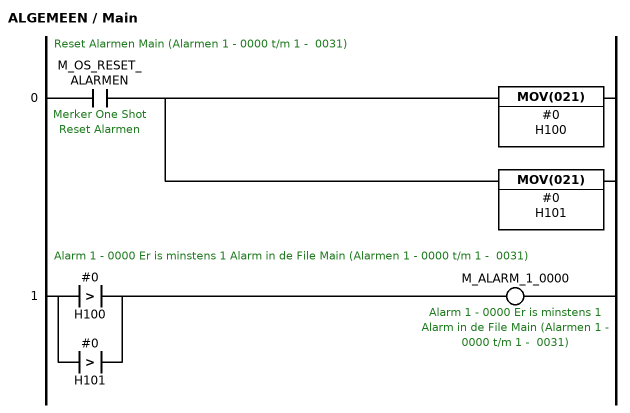
; [picture p0: ALGEMEEN / Main, rungs 0-1]
; rung 0: Reset Alarmen Main (Alarmen 1 - 0000 t/m 1 -  0031)
LD M_OS_RESET_ALARMEN  ; Merker One Shot Reset Alarmen
MOV(021) #0 H100
MOV(021) #0 H101
; rung 1: Alarm 1 - 0000 Er is minstens 1 Alarm in de File Main (Alarmen 1 - 0000 t/m 1 -  0031)
LD>(320) #0 H100
OR>(320) #0 H101
OUT M_ALARM_1_0000  ; Alarm 1 - 0000 Er is minstens 1 Alarm in de File Main (Alarmen 1 - 0000 t/m 1 -  0031)

### Section Control_Link

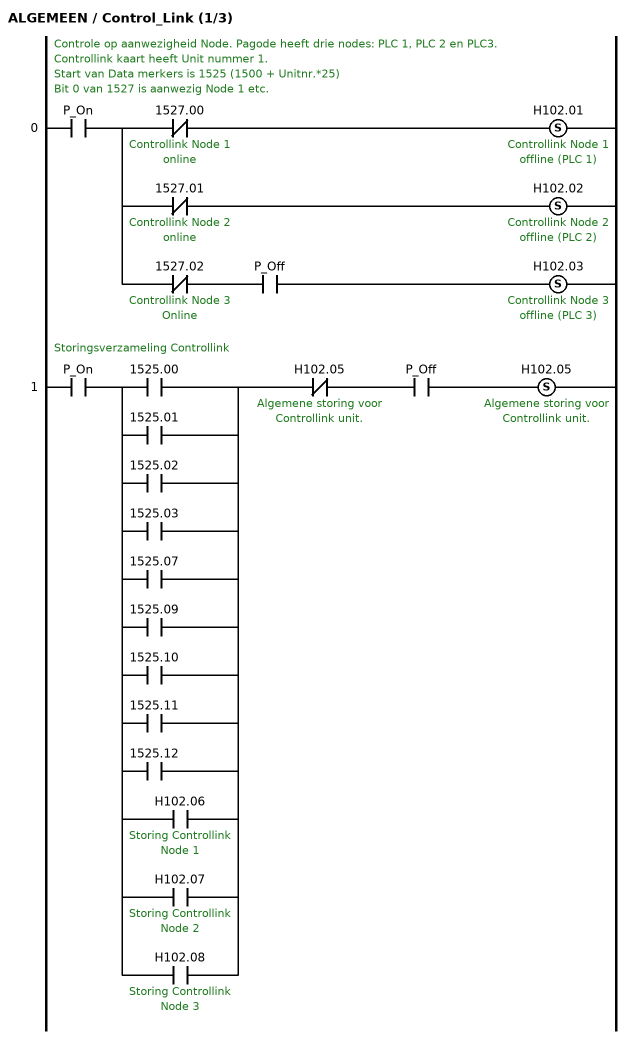
; rung 0: Controle op aanwezigheid Node. Pagode heeft drie nodes: PLC 1, PLC 2 en PLC3. / Controllink kaart heeft Unit nummer 1. / Start van Data merkers is 1525 (1500 + Unitnr.*25) / Bit 0 van 1527 is aanwezig Node 1 etc.
LD P_On
OUT TR0
ANDNOT 1527.00  ; Controllink Node 1 online
SET H102.01  ; Controllink Node 1 offline (PLC 1)
LD TR0
ANDNOT 1527.01  ; Controllink Node 2 online
SET H102.02  ; Controllink Node 2 offline (PLC 2)
LD TR0
ANDNOT 1527.02  ; Controllink Node 3 Online
AND P_Off
SET H102.03  ; Controllink Node 3 offline (PLC 3)
; rung 1: Storingsverzameling Controllink
LD P_On
LD 1525.00
OR 1525.01
OR 1525.02
OR 1525.03
OR 1525.07
OR 1525.09
OR 1525.10
OR 1525.11
OR 1525.12
OR H102.06  ; Storing Controllink Node 1
OR H102.07  ; Storing Controllink Node 2
OR H102.08  ; Storing Controllink Node 3
ANDLD
ANDNOT H102.05  ; Algemene storing voor Controllink unit.
AND P_Off
SET H102.05  ; Algemene storing voor Controllink unit.

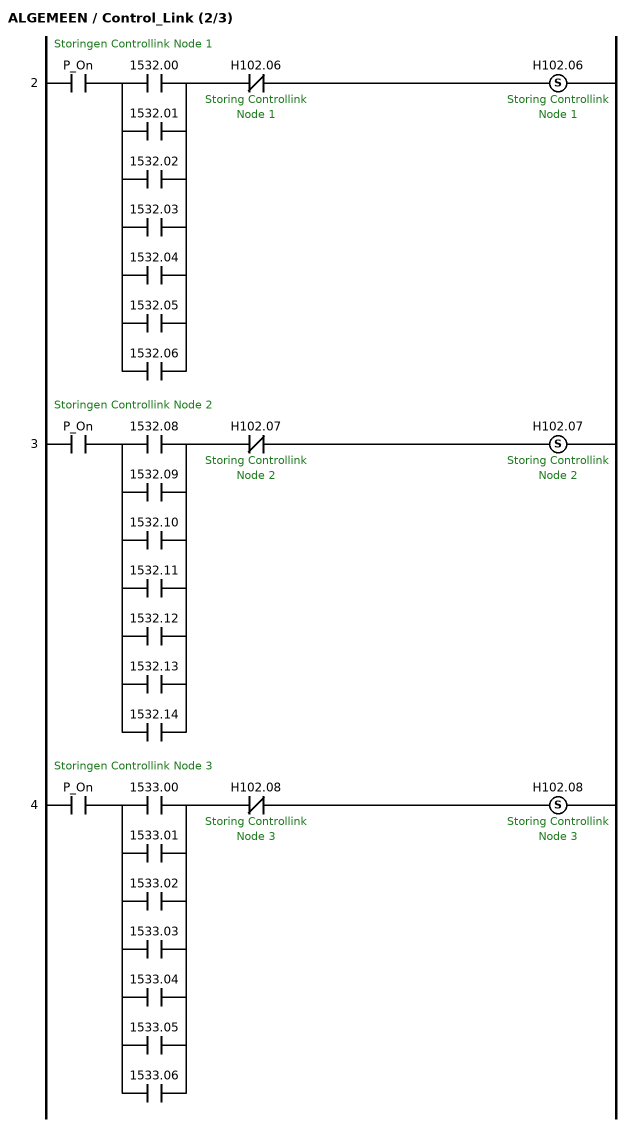
; rung 2: Storingen Controllink Node 1
LD P_On
LD 1532.00
OR 1532.01
OR 1532.02
OR 1532.03
OR 1532.04
OR 1532.05
OR 1532.06
ANDLD
ANDNOT H102.06  ; Storing Controllink Node 1
SET H102.06  ; Storing Controllink Node 1
; rung 3: Storingen Controllink Node 2
LD P_On
LD 1532.08
OR 1532.09
OR 1532.10
OR 1532.11
OR 1532.12
OR 1532.13
OR 1532.14
ANDLD
ANDNOT H102.07  ; Storing Controllink Node 2
SET H102.07  ; Storing Controllink Node 2
; rung 4: Storingen Controllink Node 3
LD P_On
LD 1533.00
OR 1533.01
OR 1533.02
OR 1533.03
OR 1533.04
OR 1533.05
OR 1533.06
ANDLD
ANDNOT H102.08  ; Storing Controllink Node 3
SET H102.08  ; Storing Controllink Node 3

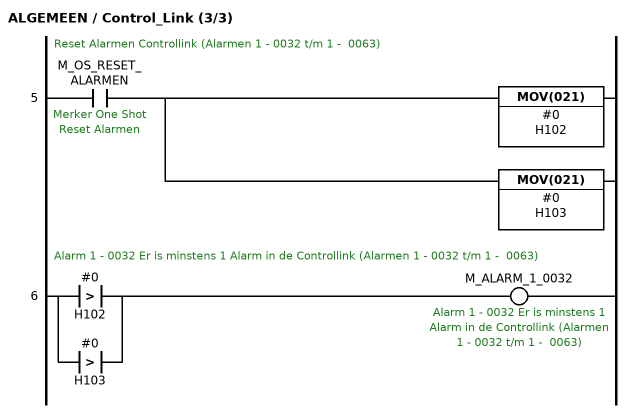
; rung 5: Reset Alarmen Controllink (Alarmen 1 - 0032 t/m 1 -  0063)
LD M_OS_RESET_ALARMEN  ; Merker One Shot Reset Alarmen
MOV(021) #0 H102
MOV(021) #0 H103
; rung 6: Alarm 1 - 0032 Er is minstens 1 Alarm in de Controllink (Alarmen 1 - 0032 t/m 1 -  0063)
LD>(320) #0 H102
OR>(320) #0 H103
OUT M_ALARM_1_0032  ; Alarm 1 - 0032 Er is minstens 1 Alarm in de Controllink (Alarmen 1 - 0032 t/m 1 -  0063)

### Section Device_Net

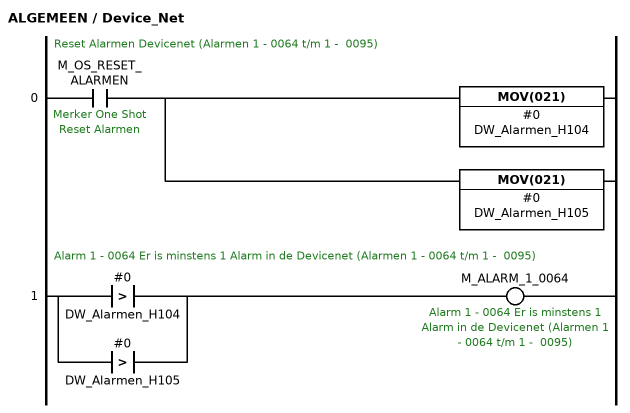
; rung 0: Reset Alarmen Devicenet (Alarmen 1 - 0064 t/m 1 -  0095)
LD M_OS_RESET_ALARMEN  ; Merker One Shot Reset Alarmen
MOV(021) #0 DW_Alarmen_H104
MOV(021) #0 DW_Alarmen_H105
; rung 1: Alarm 1 - 0064 Er is minstens 1 Alarm in de Devicenet (Alarmen 1 - 0064 t/m 1 -  0095)
LD>(320) #0 DW_Alarmen_H104
OR>(320) #0 DW_Alarmen_H105
OUT M_ALARM_1_0064  ; Alarm 1 - 0064 Er is minstens 1 Alarm in de Devicenet (Alarmen 1 - 0064 t/m 1 -  0095)

### Section Data_Opslag

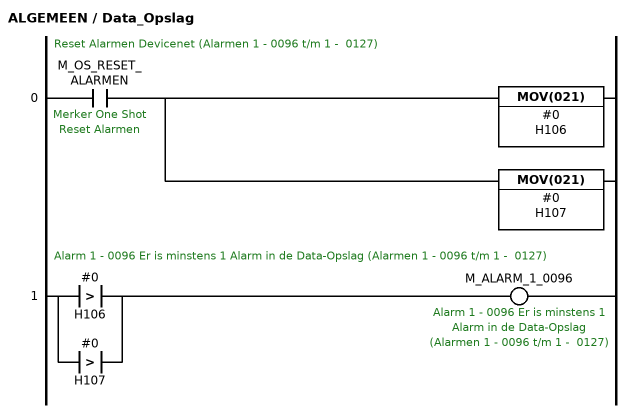
; rung 0: Reset Alarmen Devicenet (Alarmen 1 - 0096 t/m 1 -  0127)
LD M_OS_RESET_ALARMEN  ; Merker One Shot Reset Alarmen
MOV(021) #0 H106
MOV(021) #0 H107
; rung 1: Alarm 1 - 0096 Er is minstens 1 Alarm in de Data-Opslag (Alarmen 1 - 0096 t/m 1 -  0127)
LD>(320) #0 H106
OR>(320) #0 H107
OUT M_ALARM_1_0096  ; Alarm 1 - 0096 Er is minstens 1 Alarm in de Data-Opslag (Alarmen 1 - 0096 t/m 1 -  0127)

### Section Voedingen

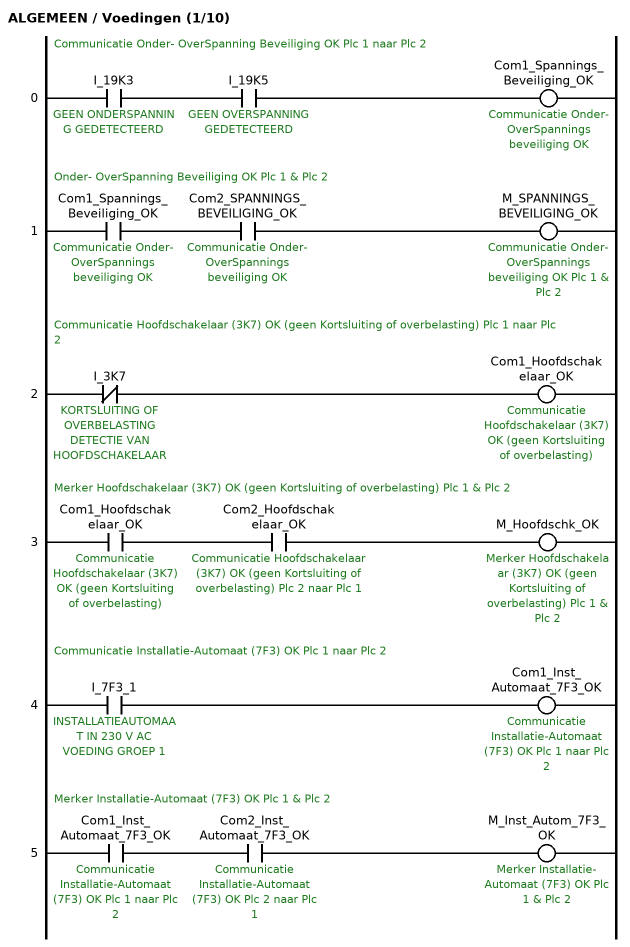
; rung 0: Communicatie Onder- OverSpanning Beveiliging OK Plc 1 naar Plc 2
LD I_19K3  ; GEEN ONDERSPANNING GEDETECTEERD
AND I_19K5  ; GEEN OVERSPANNING GEDETECTEERD
OUT Com1_Spannings_Beveiliging_OK  ; Communicatie Onder- OverSpannings beveiliging OK
; rung 1: Onder- OverSpanning Beveiliging OK Plc 1 & Plc 2
LD Com1_Spannings_Beveiliging_OK  ; Communicatie Onder- OverSpannings beveiliging OK
AND Com2_SPANNINGS_BEVEILIGING_OK  ; Communicatie Onder- OverSpannings beveiliging OK
OUT M_SPANNINGS_BEVEILIGING_OK  ; Communicatie Onder- OverSpannings beveiliging OK Plc 1 & Plc 2
; rung 2: Communicatie Hoofdschakelaar (3K7) OK (geen Kortsluiting of overbelasting) Plc 1 naar Plc 2
LDNOT I_3K7  ; KORTSLUITING OF OVERBELASTING DETECTIE VAN HOOFDSCHAKELAAR
OUT Com1_Hoofdschakelaar_OK  ; Communicatie Hoofdschakelaar (3K7) OK (geen Kortsluiting of overbelasting)
; rung 3: Merker Hoofdschakelaar (3K7) OK (geen Kortsluiting of overbelasting) Plc 1 & Plc 2
LD Com1_Hoofdschakelaar_OK  ; Communicatie Hoofdschakelaar (3K7) OK (geen Kortsluiting of overbelasting)
AND Com2_Hoofdschakelaar_OK  ; Communicatie Hoofdschakelaar (3K7) OK (geen Kortsluiting of overbelasting) Plc 2 naar Plc 1
OUT M_Hoofdschk_OK  ; Merker Hoofdschakelaar (3K7) OK (geen Kortsluiting of overbelasting) Plc 1 & Plc 2
; rung 4: Communicatie Installatie-Automaat (7F3) OK Plc 1 naar Plc 2
LD I_7F3_1  ; INSTALLATIEAUTOMAAT IN 230 V AC VOEDING GROEP 1
OUT Com1_Inst_Automaat_7F3_OK  ; Communicatie Installatie-Automaat (7F3) OK Plc 1 naar Plc 2
; rung 5: Merker Installatie-Automaat (7F3) OK Plc 1 & Plc 2
LD Com1_Inst_Automaat_7F3_OK  ; Communicatie Installatie-Automaat (7F3) OK Plc 1 naar Plc 2
AND Com2_Inst_Automaat_7F3_OK  ; Communicatie Installatie-Automaat (7F3) OK Plc 2 naar Plc 1
OUT M_Inst_Autom_7F3_OK  ; Merker Installatie-Automaat (7F3) OK Plc 1 & Plc 2

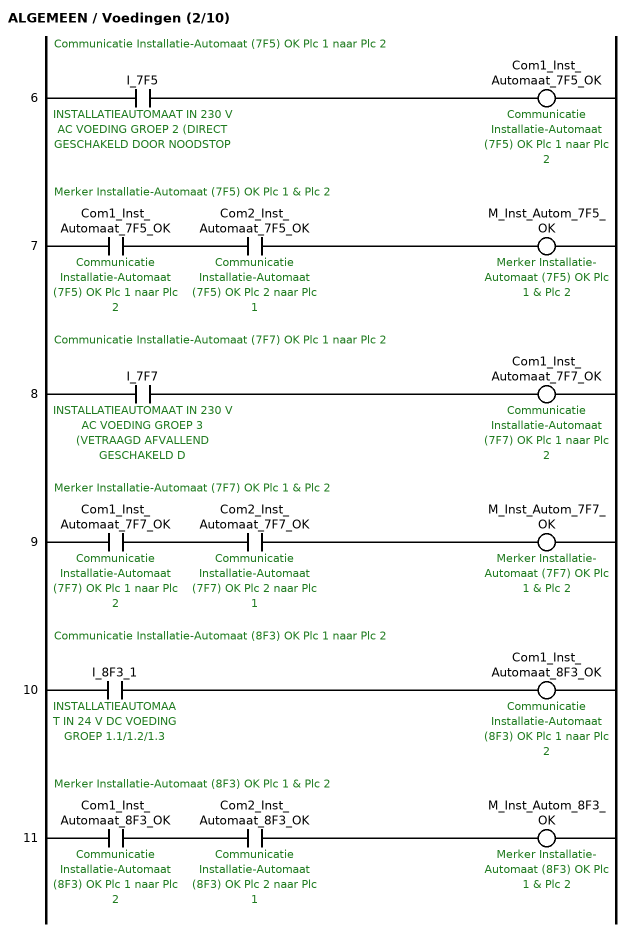
; rung 6: Communicatie Installatie-Automaat (7F5) OK Plc 1 naar Plc 2
LD I_7F5  ; INSTALLATIEAUTOMAAT IN 230 V AC VOEDING GROEP 2 (DIRECT GESCHAKELD DOOR NOODSTOP
OUT Com1_Inst_Automaat_7F5_OK  ; Communicatie Installatie-Automaat (7F5) OK Plc 1 naar Plc 2
; rung 7: Merker Installatie-Automaat (7F5) OK Plc 1 & Plc 2
LD Com1_Inst_Automaat_7F5_OK  ; Communicatie Installatie-Automaat (7F5) OK Plc 1 naar Plc 2
AND Com2_Inst_Automaat_7F5_OK  ; Communicatie Installatie-Automaat (7F5) OK Plc 2 naar Plc 1
OUT M_Inst_Autom_7F5_OK  ; Merker Installatie-Automaat (7F5) OK Plc 1 & Plc 2
; rung 8: Communicatie Installatie-Automaat (7F7) OK Plc 1 naar Plc 2
LD I_7F7  ; INSTALLATIEAUTOMAAT IN 230 V AC VOEDING GROEP 3 (VETRAAGD AFVALLEND GESCHAKELD D
OUT Com1_Inst_Automaat_7F7_OK  ; Communicatie Installatie-Automaat (7F7) OK Plc 1 naar Plc 2
; rung 9: Merker Installatie-Automaat (7F7) OK Plc 1 & Plc 2
LD Com1_Inst_Automaat_7F7_OK  ; Communicatie Installatie-Automaat (7F7) OK Plc 1 naar Plc 2
AND Com2_Inst_Automaat_7F7_OK  ; Communicatie Installatie-Automaat (7F7) OK Plc 2 naar Plc 1
OUT M_Inst_Autom_7F7_OK  ; Merker Installatie-Automaat (7F7) OK Plc 1 & Plc 2
; rung 10: Communicatie Installatie-Automaat (8F3) OK Plc 1 naar Plc 2
LD I_8F3_1  ; INSTALLATIEAUTOMAAT IN 24 V DC VOEDING GROEP 1.1/1.2/1.3
OUT Com1_Inst_Automaat_8F3_OK  ; Communicatie Installatie-Automaat (8F3) OK Plc 1 naar Plc 2
; rung 11: Merker Installatie-Automaat (8F3) OK Plc 1 & Plc 2
LD Com1_Inst_Automaat_8F3_OK  ; Communicatie Installatie-Automaat (8F3) OK Plc 1 naar Plc 2
AND Com2_Inst_Automaat_8F3_OK  ; Communicatie Installatie-Automaat (8F3) OK Plc 2 naar Plc 1
OUT M_Inst_Autom_8F3_OK  ; Merker Installatie-Automaat (8F3) OK Plc 1 & Plc 2

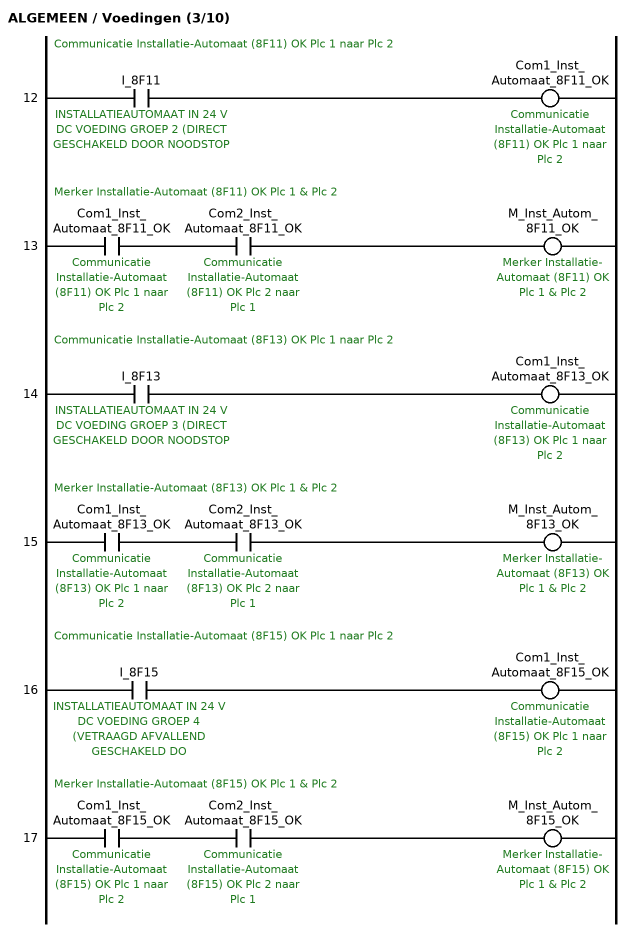
; rung 12: Communicatie Installatie-Automaat (8F11) OK Plc 1 naar Plc 2
LD I_8F11  ; INSTALLATIEAUTOMAAT IN 24 V DC VOEDING GROEP 2 (DIRECT GESCHAKELD DOOR NOODSTOP
OUT Com1_Inst_Automaat_8F11_OK  ; Communicatie Installatie-Automaat (8F11) OK Plc 1 naar Plc 2
; rung 13: Merker Installatie-Automaat (8F11) OK Plc 1 & Plc 2
LD Com1_Inst_Automaat_8F11_OK  ; Communicatie Installatie-Automaat (8F11) OK Plc 1 naar Plc 2
AND Com2_Inst_Automaat_8F11_OK  ; Communicatie Installatie-Automaat (8F11) OK Plc 2 naar Plc 1
OUT M_Inst_Autom_8F11_OK  ; Merker Installatie-Automaat (8F11) OK Plc 1 & Plc 2
; rung 14: Communicatie Installatie-Automaat (8F13) OK Plc 1 naar Plc 2
LD I_8F13  ; INSTALLATIEAUTOMAAT IN 24 V DC VOEDING GROEP 3 (DIRECT GESCHAKELD DOOR NOODSTOP
OUT Com1_Inst_Automaat_8F13_OK  ; Communicatie Installatie-Automaat (8F13) OK Plc 1 naar Plc 2
; rung 15: Merker Installatie-Automaat (8F13) OK Plc 1 & Plc 2
LD Com1_Inst_Automaat_8F13_OK  ; Communicatie Installatie-Automaat (8F13) OK Plc 1 naar Plc 2
AND Com2_Inst_Automaat_8F13_OK  ; Communicatie Installatie-Automaat (8F13) OK Plc 2 naar Plc 1
OUT M_Inst_Autom_8F13_OK  ; Merker Installatie-Automaat (8F13) OK Plc 1 & Plc 2
; rung 16: Communicatie Installatie-Automaat (8F15) OK Plc 1 naar Plc 2
LD I_8F15  ; INSTALLATIEAUTOMAAT IN 24 V DC VOEDING GROEP 4 (VETRAAGD AFVALLEND GESCHAKELD DO
OUT Com1_Inst_Automaat_8F15_OK  ; Communicatie Installatie-Automaat (8F15) OK Plc 1 naar Plc 2
; rung 17: Merker Installatie-Automaat (8F15) OK Plc 1 & Plc 2
LD Com1_Inst_Automaat_8F15_OK  ; Communicatie Installatie-Automaat (8F15) OK Plc 1 naar Plc 2
AND Com2_Inst_Automaat_8F15_OK  ; Communicatie Installatie-Automaat (8F15) OK Plc 2 naar Plc 1
OUT M_Inst_Autom_8F15_OK  ; Merker Installatie-Automaat (8F15) OK Plc 1 & Plc 2

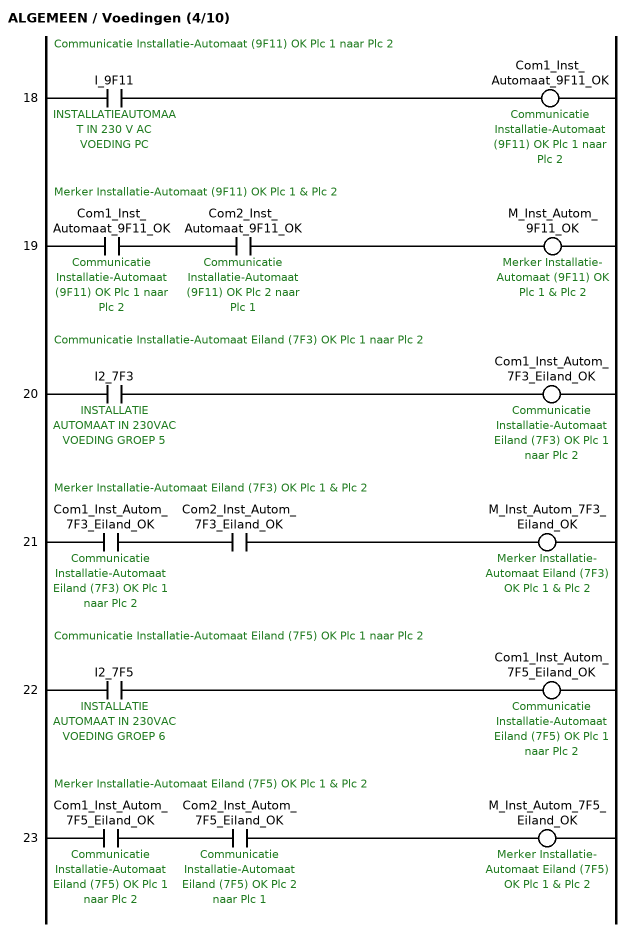
; rung 18: Communicatie Installatie-Automaat (9F11) OK Plc 1 naar Plc 2
LD I_9F11  ; INSTALLATIEAUTOMAAT IN 230 V AC VOEDING PC
OUT Com1_Inst_Automaat_9F11_OK  ; Communicatie Installatie-Automaat (9F11) OK Plc 1 naar Plc 2
; rung 19: Merker Installatie-Automaat (9F11) OK Plc 1 & Plc 2
LD Com1_Inst_Automaat_9F11_OK  ; Communicatie Installatie-Automaat (9F11) OK Plc 1 naar Plc 2
AND Com2_Inst_Automaat_9F11_OK  ; Communicatie Installatie-Automaat (9F11) OK Plc 2 naar Plc 1
OUT M_Inst_Autom_9F11_OK  ; Merker Installatie-Automaat (9F11) OK Plc 1 & Plc 2
; rung 20: Communicatie Installatie-Automaat Eiland (7F3) OK Plc 1 naar Plc 2
LD I2_7F3  ; INSTALLATIE AUTOMAAT IN 230VAC VOEDING GROEP 5
OUT Com1_Inst_Autom_7F3_Eiland_OK  ; Communicatie Installatie-Automaat Eiland (7F3) OK Plc 1 naar Plc 2
; rung 21: Merker Installatie-Automaat Eiland (7F3) OK Plc 1 & Plc 2
LD Com1_Inst_Autom_7F3_Eiland_OK  ; Communicatie Installatie-Automaat Eiland (7F3) OK Plc 1 naar Plc 2
AND Com2_Inst_Autom_7F3_Eiland_OK
OUT M_Inst_Autom_7F3_Eiland_OK  ; Merker Installatie-Automaat Eiland (7F3) OK Plc 1 & Plc 2
; rung 22: Communicatie Installatie-Automaat Eiland (7F5) OK Plc 1 naar Plc 2
LD I2_7F5  ; INSTALLATIE AUTOMAAT IN 230VAC VOEDING GROEP 6
OUT Com1_Inst_Autom_7F5_Eiland_OK  ; Communicatie Installatie-Automaat Eiland (7F5) OK Plc 1 naar Plc 2
; rung 23: Merker Installatie-Automaat Eiland (7F5) OK Plc 1 & Plc 2
LD Com1_Inst_Autom_7F5_Eiland_OK  ; Communicatie Installatie-Automaat Eiland (7F5) OK Plc 1 naar Plc 2
AND Com2_Inst_Autom_7F5_Eiland_OK  ; Communicatie Installatie-Automaat Eiland (7F5) OK Plc 2 naar Plc 1
OUT M_Inst_Autom_7F5_Eiland_OK  ; Merker Installatie-Automaat Eiland (7F5) OK Plc 1 & Plc 2

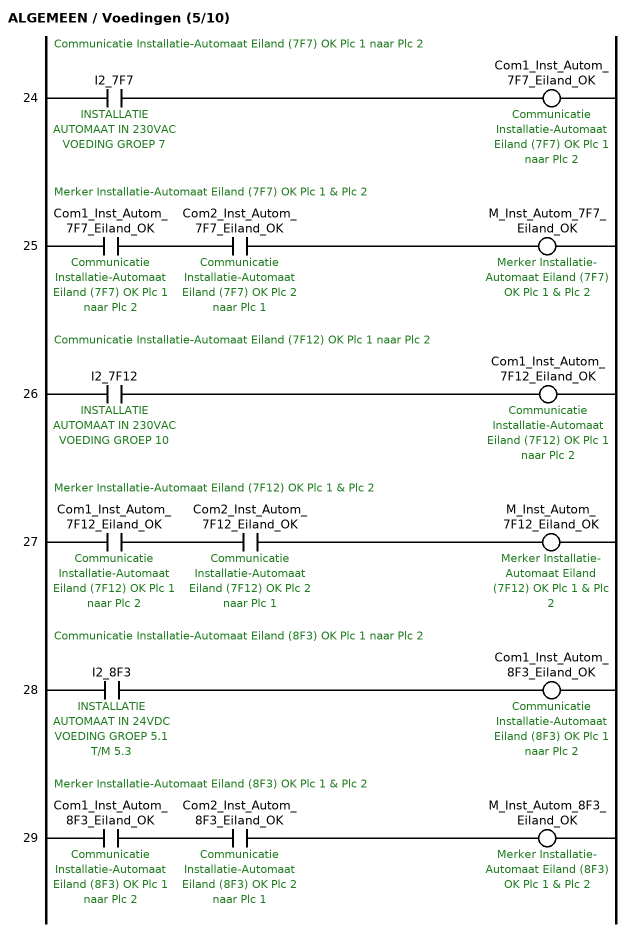
; rung 24: Communicatie Installatie-Automaat Eiland (7F7) OK Plc 1 naar Plc 2
LD I2_7F7  ; INSTALLATIE AUTOMAAT IN 230VAC VOEDING GROEP 7
OUT Com1_Inst_Autom_7F7_Eiland_OK  ; Communicatie Installatie-Automaat Eiland (7F7) OK Plc 1 naar Plc 2
; rung 25: Merker Installatie-Automaat Eiland (7F7) OK Plc 1 & Plc 2
LD Com1_Inst_Autom_7F7_Eiland_OK  ; Communicatie Installatie-Automaat Eiland (7F7) OK Plc 1 naar Plc 2
AND Com2_Inst_Autom_7F7_Eiland_OK  ; Communicatie Installatie-Automaat Eiland (7F7) OK Plc 2 naar Plc 1
OUT M_Inst_Autom_7F7_Eiland_OK  ; Merker Installatie-Automaat Eiland (7F7) OK Plc 1 & Plc 2
; rung 26: Communicatie Installatie-Automaat Eiland (7F12) OK Plc 1 naar Plc 2
LD I2_7F12  ; INSTALLATIE AUTOMAAT IN 230VAC VOEDING GROEP 10
OUT Com1_Inst_Autom_7F12_Eiland_OK  ; Communicatie Installatie-Automaat Eiland (7F12) OK Plc 1 naar Plc 2
; rung 27: Merker Installatie-Automaat Eiland (7F12) OK Plc 1 & Plc 2
LD Com1_Inst_Autom_7F12_Eiland_OK  ; Communicatie Installatie-Automaat Eiland (7F12) OK Plc 1 naar Plc 2
AND Com2_Inst_Autom_7F12_Eiland_OK  ; Communicatie Installatie-Automaat Eiland (7F12) OK Plc 2 naar Plc 1
OUT M_Inst_Autom_7F12_Eiland_OK  ; Merker Installatie-Automaat Eiland (7F12) OK Plc 1 & Plc 2
; rung 28: Communicatie Installatie-Automaat Eiland (8F3) OK Plc 1 naar Plc 2
LD I2_8F3  ; INSTALLATIE AUTOMAAT IN 24VDC VOEDING GROEP 5.1 T/M 5.3
OUT Com1_Inst_Autom_8F3_Eiland_OK  ; Communicatie Installatie-Automaat Eiland (8F3) OK Plc 1 naar Plc 2
; rung 29: Merker Installatie-Automaat Eiland (8F3) OK Plc 1 & Plc 2
LD Com1_Inst_Autom_8F3_Eiland_OK  ; Communicatie Installatie-Automaat Eiland (8F3) OK Plc 1 naar Plc 2
AND Com2_Inst_Autom_8F3_Eiland_OK  ; Communicatie Installatie-Automaat Eiland (8F3) OK Plc 2 naar Plc 1
OUT M_Inst_Autom_8F3_Eiland_OK  ; Merker Installatie-Automaat Eiland (8F3) OK Plc 1 & Plc 2

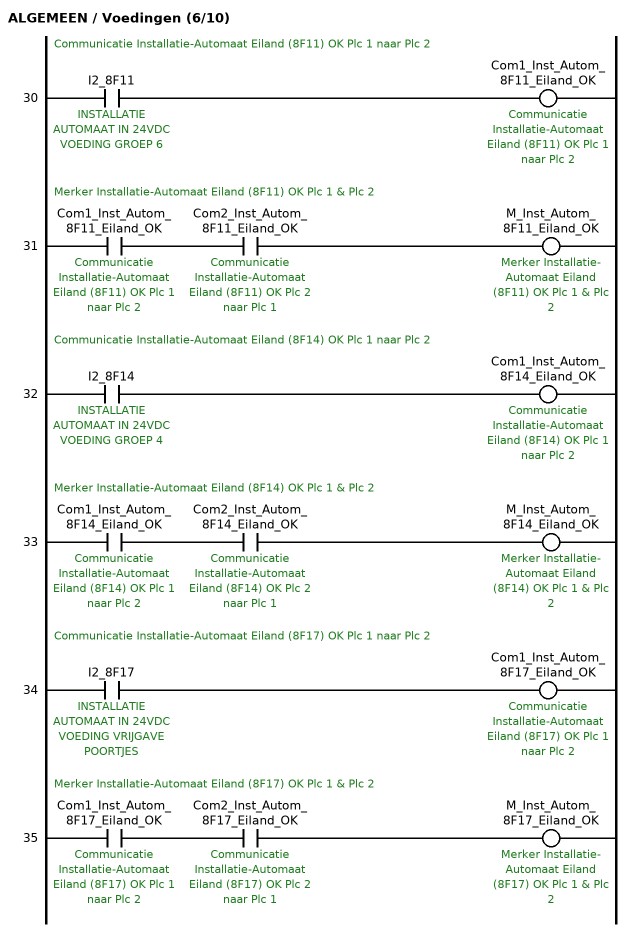
; rung 30: Communicatie Installatie-Automaat Eiland (8F11) OK Plc 1 naar Plc 2
LD I2_8F11  ; INSTALLATIE AUTOMAAT IN 24VDC VOEDING GROEP 6
OUT Com1_Inst_Autom_8F11_Eiland_OK  ; Communicatie Installatie-Automaat Eiland (8F11) OK Plc 1 naar Plc 2
; rung 31: Merker Installatie-Automaat Eiland (8F11) OK Plc 1 & Plc 2
LD Com1_Inst_Autom_8F11_Eiland_OK  ; Communicatie Installatie-Automaat Eiland (8F11) OK Plc 1 naar Plc 2
AND Com2_Inst_Autom_8F11_Eiland_OK  ; Communicatie Installatie-Automaat Eiland (8F11) OK Plc 2 naar Plc 1
OUT M_Inst_Autom_8F11_Eiland_OK  ; Merker Installatie-Automaat Eiland (8F11) OK Plc 1 & Plc 2
; rung 32: Communicatie Installatie-Automaat Eiland (8F14) OK Plc 1 naar Plc 2
LD I2_8F14  ; INSTALLATIE AUTOMAAT IN 24VDC VOEDING GROEP 4
OUT Com1_Inst_Autom_8F14_Eiland_OK  ; Communicatie Installatie-Automaat Eiland (8F14) OK Plc 1 naar Plc 2
; rung 33: Merker Installatie-Automaat Eiland (8F14) OK Plc 1 & Plc 2
LD Com1_Inst_Autom_8F14_Eiland_OK  ; Communicatie Installatie-Automaat Eiland (8F14) OK Plc 1 naar Plc 2
AND Com2_Inst_Autom_8F14_Eiland_OK  ; Communicatie Installatie-Automaat Eiland (8F14) OK Plc 2 naar Plc 1
OUT M_Inst_Autom_8F14_Eiland_OK  ; Merker Installatie-Automaat Eiland (8F14) OK Plc 1 & Plc 2
; rung 34: Communicatie Installatie-Automaat Eiland (8F17) OK Plc 1 naar Plc 2
LD I2_8F17  ; INSTALLATIE AUTOMAAT IN 24VDC VOEDING VRIJGAVE POORTJES
OUT Com1_Inst_Autom_8F17_Eiland_OK  ; Communicatie Installatie-Automaat Eiland (8F17) OK Plc 1 naar Plc 2
; rung 35: Merker Installatie-Automaat Eiland (8F17) OK Plc 1 & Plc 2
LD Com1_Inst_Autom_8F17_Eiland_OK  ; Communicatie Installatie-Automaat Eiland (8F17) OK Plc 1 naar Plc 2
AND Com2_Inst_Autom_8F17_Eiland_OK  ; Communicatie Installatie-Automaat Eiland (8F17) OK Plc 2 naar Plc 1
OUT M_Inst_Autom_8F17_Eiland_OK  ; Merker Installatie-Automaat Eiland (8F17) OK Plc 1 & Plc 2

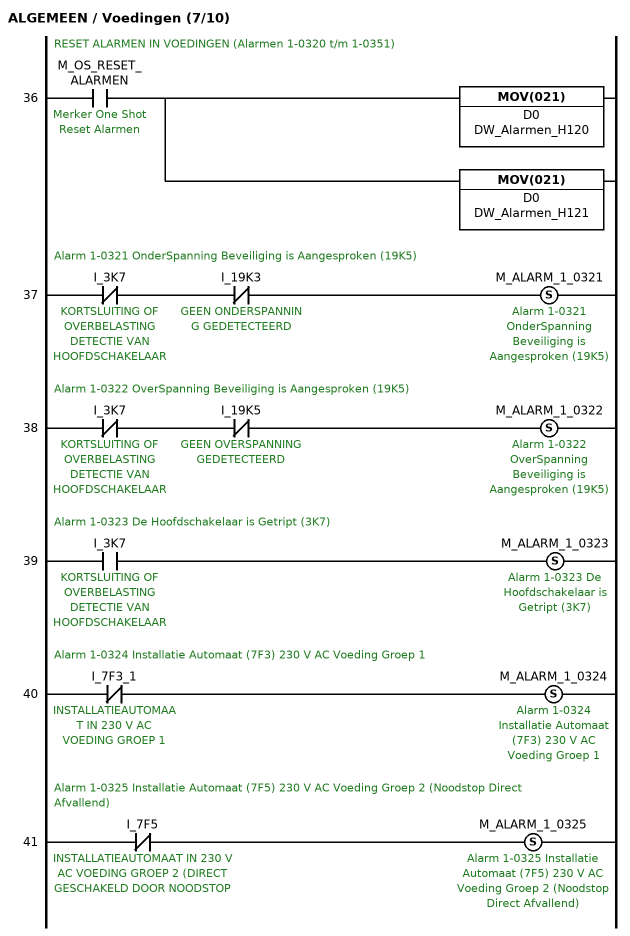
; rung 36: RESET ALARMEN IN VOEDINGEN (Alarmen 1-0320 t/m 1-0351)
LD M_OS_RESET_ALARMEN  ; Merker One Shot Reset Alarmen
MOV(021) D0 DW_Alarmen_H120
MOV(021) D0 DW_Alarmen_H121
; rung 37: Alarm 1-0321 OnderSpanning Beveiliging is Aangesproken (19K5)
LDNOT I_3K7  ; KORTSLUITING OF OVERBELASTING DETECTIE VAN HOOFDSCHAKELAAR
ANDNOT I_19K3  ; GEEN ONDERSPANNING GEDETECTEERD
SET M_ALARM_1_0321  ; Alarm 1-0321 OnderSpanning Beveiliging is Aangesproken (19K5)
; rung 38: Alarm 1-0322 OverSpanning Beveiliging is Aangesproken (19K5)
LDNOT I_3K7  ; KORTSLUITING OF OVERBELASTING DETECTIE VAN HOOFDSCHAKELAAR
ANDNOT I_19K5  ; GEEN OVERSPANNING GEDETECTEERD
SET M_ALARM_1_0322  ; Alarm 1-0322 OverSpanning Beveiliging is Aangesproken (19K5)
; rung 39: Alarm 1-0323 De Hoofdschakelaar is Getript (3K7)
LD I_3K7  ; KORTSLUITING OF OVERBELASTING DETECTIE VAN HOOFDSCHAKELAAR
SET M_ALARM_1_0323  ; Alarm 1-0323 De Hoofdschakelaar is Getript (3K7)
; rung 40: Alarm 1-0324 Installatie Automaat (7F3) 230 V AC Voeding Groep 1
LDNOT I_7F3_1  ; INSTALLATIEAUTOMAAT IN 230 V AC VOEDING GROEP 1
SET M_ALARM_1_0324  ; Alarm 1-0324 Installatie Automaat (7F3) 230 V AC Voeding Groep 1
; rung 41: Alarm 1-0325 Installatie Automaat (7F5) 230 V AC Voeding Groep 2 (Noodstop Direct Afvallend)
LDNOT I_7F5  ; INSTALLATIEAUTOMAAT IN 230 V AC VOEDING GROEP 2 (DIRECT GESCHAKELD DOOR NOODSTOP
SET M_ALARM_1_0325  ; Alarm 1-0325 Installatie Automaat (7F5) 230 V AC Voeding Groep 2 (Noodstop Direct Afvallend)

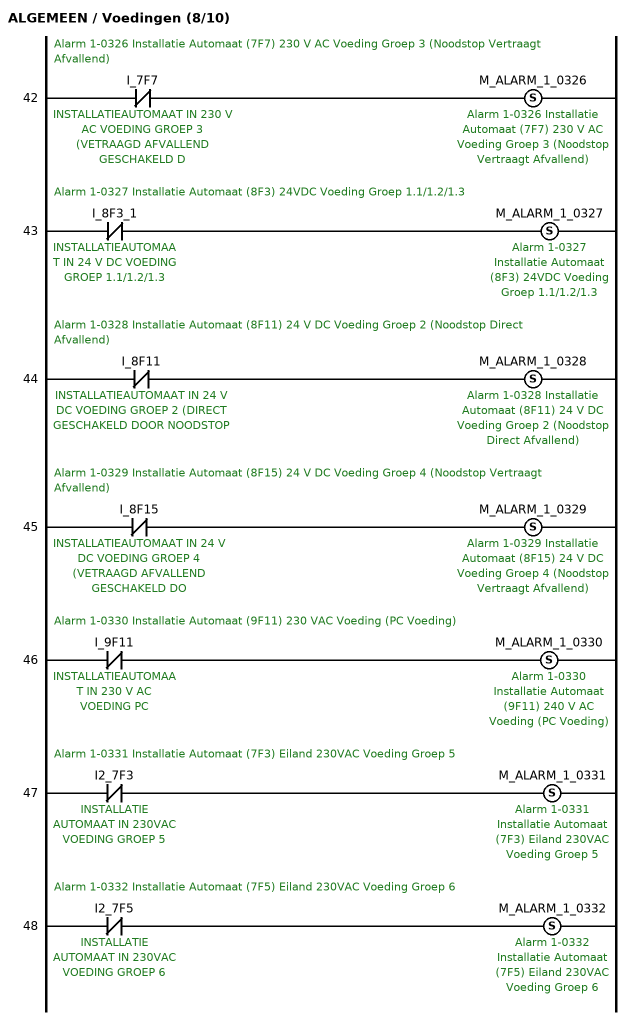
; rung 42: Alarm 1-0326 Installatie Automaat (7F7) 230 V AC Voeding Groep 3 (Noodstop Vertraagt Afvallend)
LDNOT I_7F7  ; INSTALLATIEAUTOMAAT IN 230 V AC VOEDING GROEP 3 (VETRAAGD AFVALLEND GESCHAKELD D
SET M_ALARM_1_0326  ; Alarm 1-0326 Installatie Automaat (7F7) 230 V AC Voeding Groep 3 (Noodstop Vertraagt Afvallend)
; rung 43: Alarm 1-0327 Installatie Automaat (8F3) 24VDC Voeding Groep 1.1/1.2/1.3
LDNOT I_8F3_1  ; INSTALLATIEAUTOMAAT IN 24 V DC VOEDING GROEP 1.1/1.2/1.3
SET M_ALARM_1_0327  ; Alarm 1-0327 Installatie Automaat (8F3) 24VDC Voeding Groep 1.1/1.2/1.3
; rung 44: Alarm 1-0328 Installatie Automaat (8F11) 24 V DC Voeding Groep 2 (Noodstop Direct Afvallend)
LDNOT I_8F11  ; INSTALLATIEAUTOMAAT IN 24 V DC VOEDING GROEP 2 (DIRECT GESCHAKELD DOOR NOODSTOP
SET M_ALARM_1_0328  ; Alarm 1-0328 Installatie Automaat (8F11) 24 V DC Voeding Groep 2 (Noodstop Direct Afvallend)
; rung 45: Alarm 1-0329 Installatie Automaat (8F15) 24 V DC Voeding Groep 4 (Noodstop Vertraagt Afvallend)
LDNOT I_8F15  ; INSTALLATIEAUTOMAAT IN 24 V DC VOEDING GROEP 4 (VETRAAGD AFVALLEND GESCHAKELD DO
SET M_ALARM_1_0329  ; Alarm 1-0329 Installatie Automaat (8F15) 24 V DC Voeding Groep 4 (Noodstop Vertraagt Afvallend)
; rung 46: Alarm 1-0330 Installatie Automaat (9F11) 230 VAC Voeding (PC Voeding)
LDNOT I_9F11  ; INSTALLATIEAUTOMAAT IN 230 V AC VOEDING PC
SET M_ALARM_1_0330  ; Alarm 1-0330 Installatie Automaat (9F11) 240 V AC Voeding (PC Voeding)
; rung 47: Alarm 1-0331 Installatie Automaat (7F3) Eiland 230VAC Voeding Groep 5
LDNOT I2_7F3  ; INSTALLATIE AUTOMAAT IN 230VAC VOEDING GROEP 5
SET M_ALARM_1_0331  ; Alarm 1-0331 Installatie Automaat (7F3) Eiland 230VAC Voeding Groep 5
; rung 48: Alarm 1-0332 Installatie Automaat (7F5) Eiland 230VAC Voeding Groep 6
LDNOT I2_7F5  ; INSTALLATIE AUTOMAAT IN 230VAC VOEDING GROEP 6
SET M_ALARM_1_0332  ; Alarm 1-0332 Installatie Automaat (7F5) Eiland 230VAC Voeding Groep 6

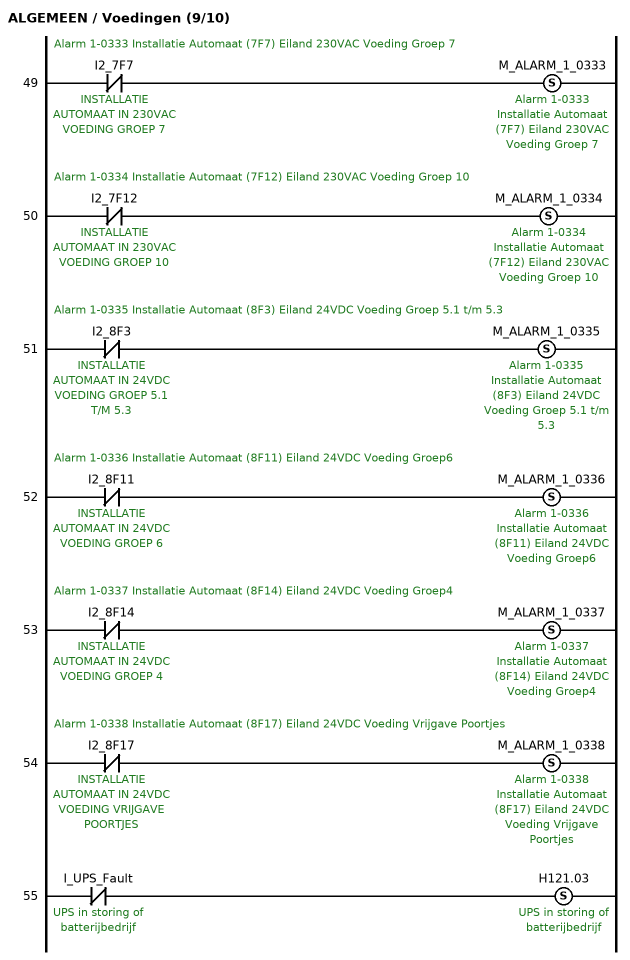
; rung 49: Alarm 1-0333 Installatie Automaat (7F7) Eiland 230VAC Voeding Groep 7
LDNOT I2_7F7  ; INSTALLATIE AUTOMAAT IN 230VAC VOEDING GROEP 7
SET M_ALARM_1_0333  ; Alarm 1-0333 Installatie Automaat (7F7) Eiland 230VAC Voeding Groep 7
; rung 50: Alarm 1-0334 Installatie Automaat (7F12) Eiland 230VAC Voeding Groep 10
LDNOT I2_7F12  ; INSTALLATIE AUTOMAAT IN 230VAC VOEDING GROEP 10
SET M_ALARM_1_0334  ; Alarm 1-0334 Installatie Automaat (7F12) Eiland 230VAC Voeding Groep 10
; rung 51: Alarm 1-0335 Installatie Automaat (8F3) Eiland 24VDC Voeding Groep 5.1 t/m 5.3
LDNOT I2_8F3  ; INSTALLATIE AUTOMAAT IN 24VDC VOEDING GROEP 5.1 T/M 5.3
SET M_ALARM_1_0335  ; Alarm 1-0335 Installatie Automaat (8F3) Eiland 24VDC Voeding Groep 5.1 t/m 5.3
; rung 52: Alarm 1-0336 Installatie Automaat (8F11) Eiland 24VDC Voeding Groep6
LDNOT I2_8F11  ; INSTALLATIE AUTOMAAT IN 24VDC VOEDING GROEP 6
SET M_ALARM_1_0336  ; Alarm 1-0336 Installatie Automaat (8F11) Eiland 24VDC Voeding Groep6
; rung 53: Alarm 1-0337 Installatie Automaat (8F14) Eiland 24VDC Voeding Groep4
LDNOT I2_8F14  ; INSTALLATIE AUTOMAAT IN 24VDC VOEDING GROEP 4
SET M_ALARM_1_0337  ; Alarm 1-0337 Installatie Automaat (8F14) Eiland 24VDC Voeding Groep4
; rung 54: Alarm 1-0338 Installatie Automaat (8F17) Eiland 24VDC Voeding Vrijgave Poortjes
LDNOT I2_8F17  ; INSTALLATIE AUTOMAAT IN 24VDC VOEDING VRIJGAVE POORTJES
SET M_ALARM_1_0338  ; Alarm 1-0338 Installatie Automaat (8F17) Eiland 24VDC Voeding Vrijgave Poortjes
; rung 55
LDNOT I_UPS_Fault  ; UPS in storing of batterijbedrijf
SET H121.03  ; UPS in storing of batterijbedrijf

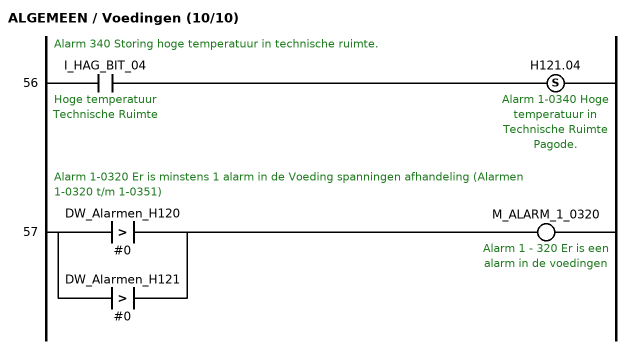
; rung 56: Alarm 340 Storing hoge temperatuur in technische ruimte.
LD I_HAG_BIT_04  ; Hoge temperatuur Technische Ruimte
SET H121.04  ; Alarm 1-0340 Hoge temperatuur in Technische Ruimte Pagode.
; rung 57: Alarm 1-0320 Er is minstens 1 alarm in de Voeding spanningen afhandeling (Alarmen 1-0320 t/m 1-0351)
LD>(320) DW_Alarmen_H120 #0
OR>(320) DW_Alarmen_H121 #0
OUT M_ALARM_1_0320  ; Alarm 1 - 320 Er is een alarm in de voedingen

### Section I_O_Controle

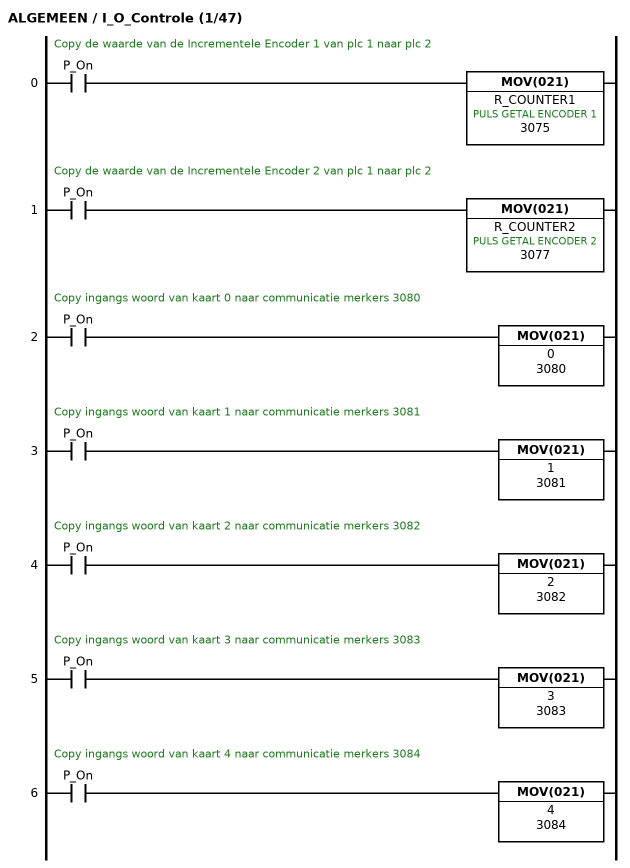
; rung 0: Copy de waarde van de Incrementele Encoder 1 van plc 1 naar plc 2
LD P_On
MOV(021) R_COUNTER1 3075  ; PULS GETAL ENCODER 1
; rung 1: Copy de waarde van de Incrementele Encoder 2 van plc 1 naar plc 2
LD P_On
MOV(021) R_COUNTER2 3077  ; PULS GETAL ENCODER 2
; rung 2: Copy ingangs woord van kaart 0 naar communicatie merkers 3080
LD P_On
MOV(021) 0 3080
; rung 3: Copy ingangs woord van kaart 1 naar communicatie merkers 3081
LD P_On
MOV(021) 1 3081
; rung 4: Copy ingangs woord van kaart 2 naar communicatie merkers 3082
LD P_On
MOV(021) 2 3082
; rung 5: Copy ingangs woord van kaart 3 naar communicatie merkers 3083
LD P_On
MOV(021) 3 3083
; rung 6: Copy ingangs woord van kaart 4 naar communicatie merkers 3084
LD P_On
MOV(021) 4 3084

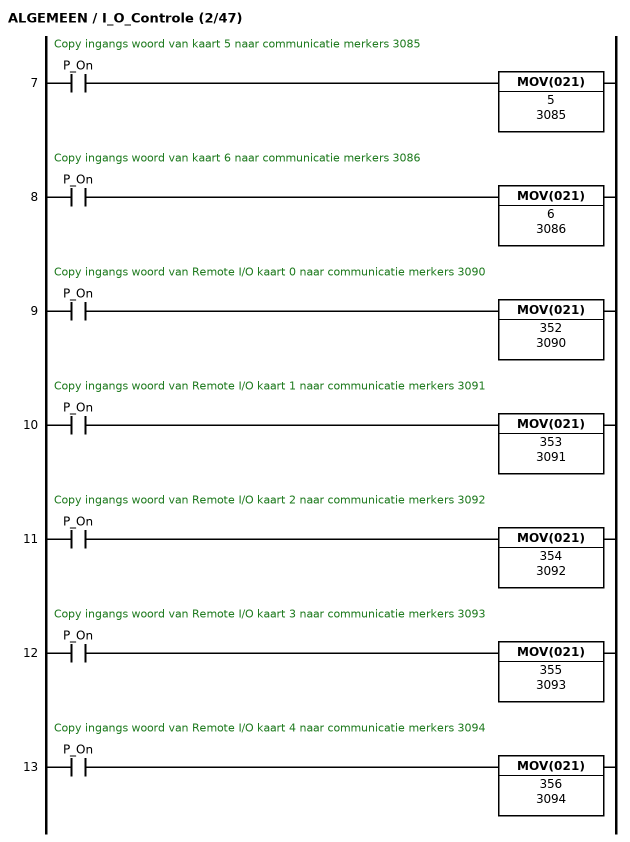
; rung 7: Copy ingangs woord van kaart 5 naar communicatie merkers 3085
LD P_On
MOV(021) 5 3085
; rung 8: Copy ingangs woord van kaart 6 naar communicatie merkers 3086
LD P_On
MOV(021) 6 3086
; rung 9: Copy ingangs woord van Remote I/O kaart 0 naar communicatie merkers 3090
LD P_On
MOV(021) 352 3090
; rung 10: Copy ingangs woord van Remote I/O kaart 1 naar communicatie merkers 3091
LD P_On
MOV(021) 353 3091
; rung 11: Copy ingangs woord van Remote I/O kaart 2 naar communicatie merkers 3092
LD P_On
MOV(021) 354 3092
; rung 12: Copy ingangs woord van Remote I/O kaart 3 naar communicatie merkers 3093
LD P_On
MOV(021) 355 3093
; rung 13: Copy ingangs woord van Remote I/O kaart 4 naar communicatie merkers 3094
LD P_On
MOV(021) 356 3094

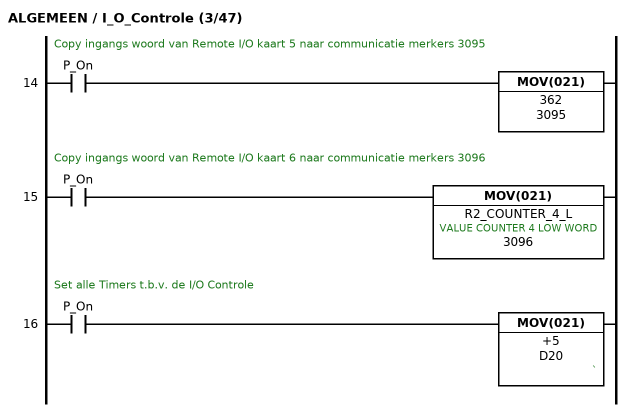
; rung 14: Copy ingangs woord van Remote I/O kaart 5 naar communicatie merkers 3095
LD P_On
MOV(021) 362 3095
; rung 15: Copy ingangs woord van Remote I/O kaart 6 naar communicatie merkers 3096
LD P_On
MOV(021) R2_COUNTER_4_L 3096  ; VALUE COUNTER 4 LOW WORD
; rung 16: Set alle Timers t.b.v. de I/O Controle
LD P_On
MOV(021) +5 D20  ; `

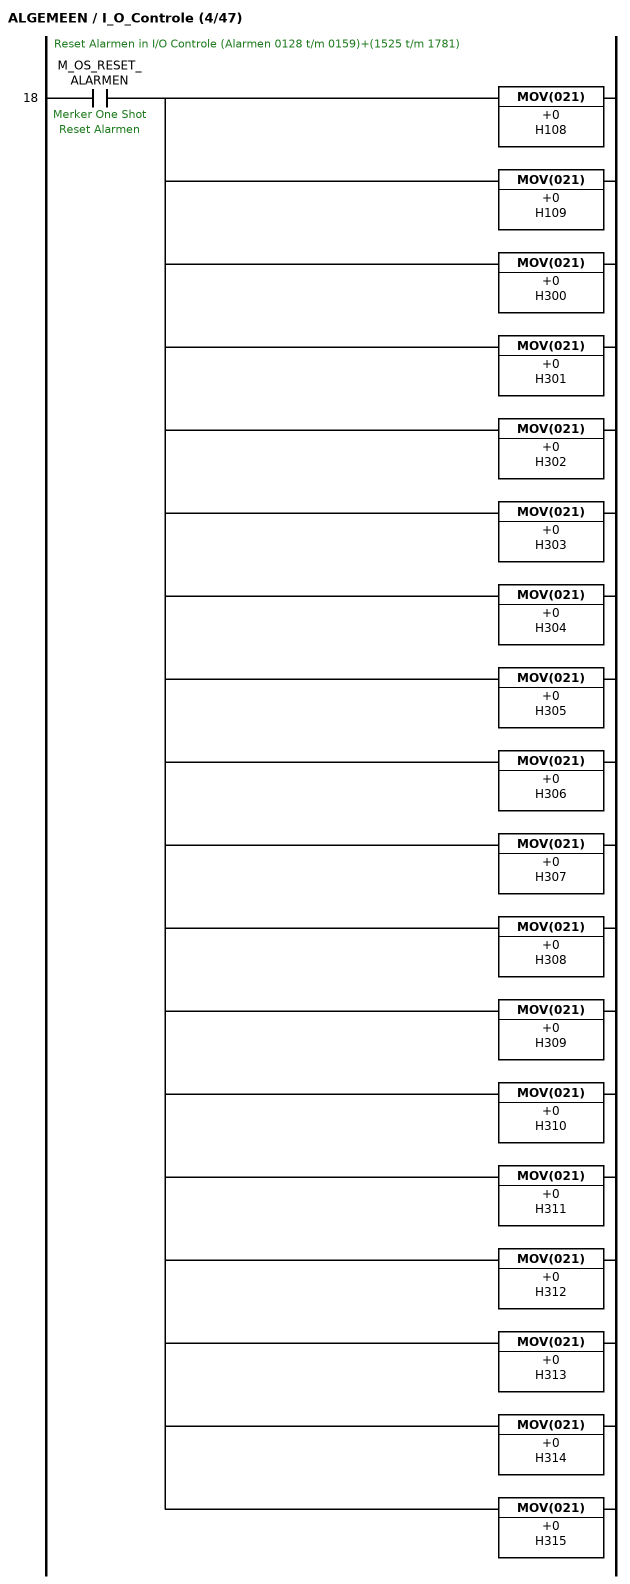
; rung 18: Reset Alarmen in I/O Controle (Alarmen 0128 t/m 0159)+(1525 t/m 1781)
LD M_OS_RESET_ALARMEN  ; Merker One Shot Reset Alarmen
MOV(021) +0 H108
MOV(021) +0 H109
MOV(021) +0 H300
MOV(021) +0 H301
MOV(021) +0 H302
MOV(021) +0 H303
MOV(021) +0 H304
MOV(021) +0 H305
MOV(021) +0 H306
MOV(021) +0 H307
MOV(021) +0 H308
MOV(021) +0 H309
MOV(021) +0 H310
MOV(021) +0 H311
MOV(021) +0 H312
MOV(021) +0 H313
MOV(021) +0 H314
MOV(021) +0 H315

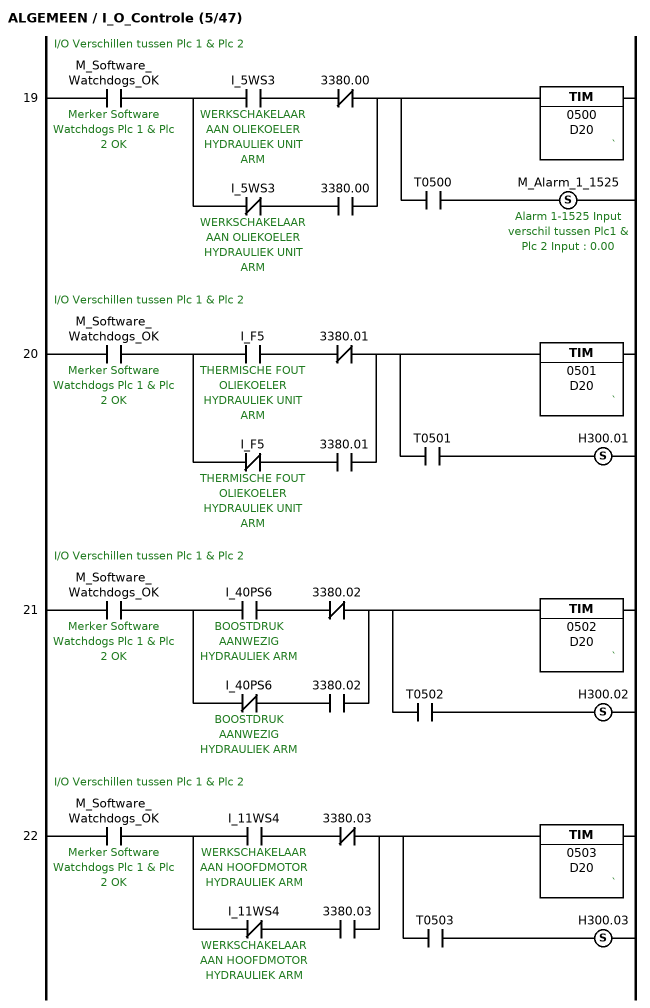
; rung 19: I/O Verschillen tussen Plc 1 & Plc 2
LD M_Software_Watchdogs_OK  ; Merker Software Watchdogs Plc 1 & Plc 2 OK
LD I_5WS3  ; WERKSCHAKELAAR AAN OLIEKOELER HYDRAULIEK UNIT ARM
ANDNOT 3380.00
LDNOT I_5WS3  ; WERKSCHAKELAAR AAN OLIEKOELER HYDRAULIEK UNIT ARM
AND 3380.00
ORLD
ANDLD
TIM 0500 D20  ; `
AND T0500
SET M_Alarm_1_1525  ; Alarm 1-1525 Input verschil tussen Plc1 & Plc 2 Input : 0.00
; rung 20: I/O Verschillen tussen Plc 1 & Plc 2
LD M_Software_Watchdogs_OK  ; Merker Software Watchdogs Plc 1 & Plc 2 OK
LD I_F5  ; THERMISCHE FOUT OLIEKOELER HYDRAULIEK UNIT ARM
ANDNOT 3380.01
LDNOT I_F5  ; THERMISCHE FOUT OLIEKOELER HYDRAULIEK UNIT ARM
AND 3380.01
ORLD
ANDLD
TIM 0501 D20  ; `
AND T0501
SET H300.01
; rung 21: I/O Verschillen tussen Plc 1 & Plc 2
LD M_Software_Watchdogs_OK  ; Merker Software Watchdogs Plc 1 & Plc 2 OK
LD I_40PS6  ; BOOSTDRUK AANWEZIG HYDRAULIEK ARM
ANDNOT 3380.02
LDNOT I_40PS6  ; BOOSTDRUK AANWEZIG HYDRAULIEK ARM
AND 3380.02
ORLD
ANDLD
TIM 0502 D20  ; `
AND T0502
SET H300.02
; rung 22: I/O Verschillen tussen Plc 1 & Plc 2
LD M_Software_Watchdogs_OK  ; Merker Software Watchdogs Plc 1 & Plc 2 OK
LD I_11WS4  ; WERKSCHAKELAAR AAN HOOFDMOTOR HYDRAULIEK ARM
ANDNOT 3380.03
LDNOT I_11WS4  ; WERKSCHAKELAAR AAN HOOFDMOTOR HYDRAULIEK ARM
AND 3380.03
ORLD
ANDLD
TIM 0503 D20  ; `
AND T0503
SET H300.03

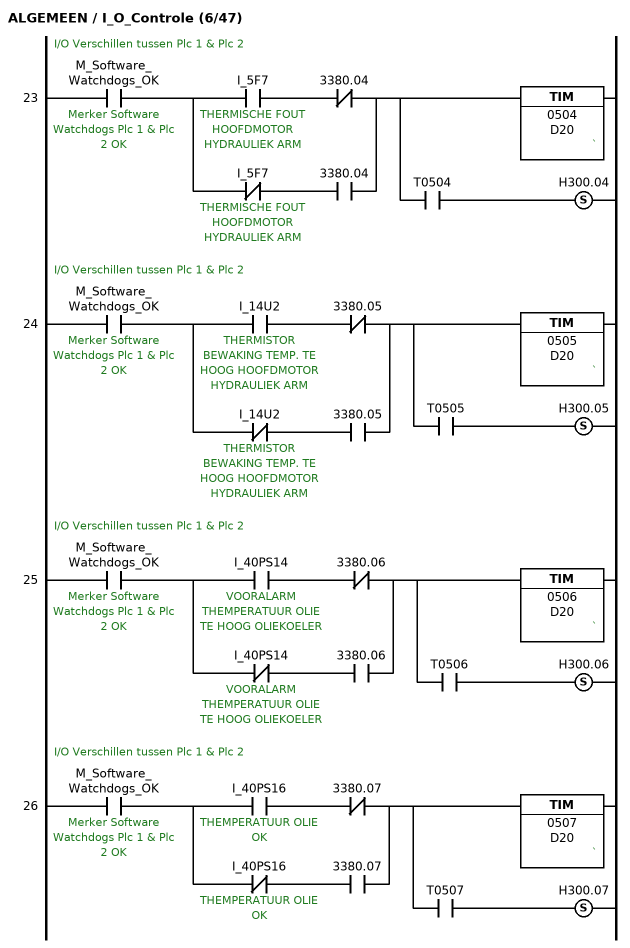
; rung 23: I/O Verschillen tussen Plc 1 & Plc 2
LD M_Software_Watchdogs_OK  ; Merker Software Watchdogs Plc 1 & Plc 2 OK
LD I_5F7  ; THERMISCHE FOUT HOOFDMOTOR HYDRAULIEK ARM
ANDNOT 3380.04
LDNOT I_5F7  ; THERMISCHE FOUT HOOFDMOTOR HYDRAULIEK ARM
AND 3380.04
ORLD
ANDLD
TIM 0504 D20  ; `
AND T0504
SET H300.04
; rung 24: I/O Verschillen tussen Plc 1 & Plc 2
LD M_Software_Watchdogs_OK  ; Merker Software Watchdogs Plc 1 & Plc 2 OK
LD I_14U2  ; THERMISTOR BEWAKING TEMP. TE HOOG HOOFDMOTOR HYDRAULIEK ARM
ANDNOT 3380.05
LDNOT I_14U2  ; THERMISTOR BEWAKING TEMP. TE HOOG HOOFDMOTOR HYDRAULIEK ARM
AND 3380.05
ORLD
ANDLD
TIM 0505 D20  ; `
AND T0505
SET H300.05
; rung 25: I/O Verschillen tussen Plc 1 & Plc 2
LD M_Software_Watchdogs_OK  ; Merker Software Watchdogs Plc 1 & Plc 2 OK
LD I_40PS14  ; VOORALARM THEMPERATUUR OLIE TE HOOG OLIEKOELER
ANDNOT 3380.06
LDNOT I_40PS14  ; VOORALARM THEMPERATUUR OLIE TE HOOG OLIEKOELER
AND 3380.06
ORLD
ANDLD
TIM 0506 D20  ; `
AND T0506
SET H300.06
; rung 26: I/O Verschillen tussen Plc 1 & Plc 2
LD M_Software_Watchdogs_OK  ; Merker Software Watchdogs Plc 1 & Plc 2 OK
LD I_40PS16  ; THEMPERATUUR OLIE OK
ANDNOT 3380.07
LDNOT I_40PS16  ; THEMPERATUUR OLIE OK
AND 3380.07
ORLD
ANDLD
TIM 0507 D20  ; `
AND T0507
SET H300.07

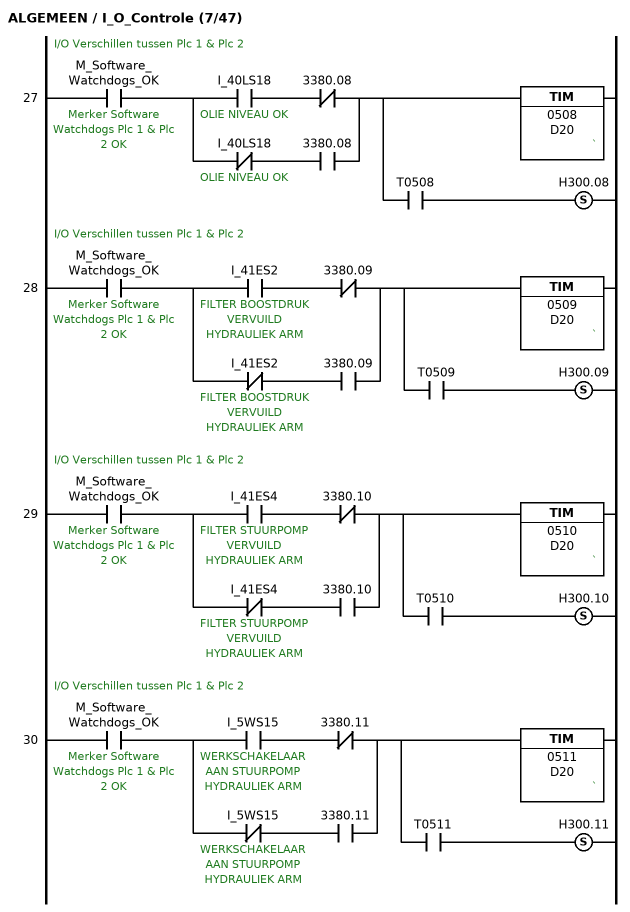
; rung 27: I/O Verschillen tussen Plc 1 & Plc 2
LD M_Software_Watchdogs_OK  ; Merker Software Watchdogs Plc 1 & Plc 2 OK
LD I_40LS18  ; OLIE NIVEAU OK
ANDNOT 3380.08
LDNOT I_40LS18  ; OLIE NIVEAU OK
AND 3380.08
ORLD
ANDLD
TIM 0508 D20  ; `
AND T0508
SET H300.08
; rung 28: I/O Verschillen tussen Plc 1 & Plc 2
LD M_Software_Watchdogs_OK  ; Merker Software Watchdogs Plc 1 & Plc 2 OK
LD I_41ES2  ; FILTER BOOSTDRUK VERVUILD HYDRAULIEK ARM
ANDNOT 3380.09
LDNOT I_41ES2  ; FILTER BOOSTDRUK VERVUILD HYDRAULIEK ARM
AND 3380.09
ORLD
ANDLD
TIM 0509 D20  ; `
AND T0509
SET H300.09
; rung 29: I/O Verschillen tussen Plc 1 & Plc 2
LD M_Software_Watchdogs_OK  ; Merker Software Watchdogs Plc 1 & Plc 2 OK
LD I_41ES4  ; FILTER STUURPOMP VERVUILD HYDRAULIEK ARM
ANDNOT 3380.10
LDNOT I_41ES4  ; FILTER STUURPOMP VERVUILD HYDRAULIEK ARM
AND 3380.10
ORLD
ANDLD
TIM 0510 D20  ; `
AND T0510
SET H300.10
; rung 30: I/O Verschillen tussen Plc 1 & Plc 2
LD M_Software_Watchdogs_OK  ; Merker Software Watchdogs Plc 1 & Plc 2 OK
LD I_5WS15  ; WERKSCHAKELAAR AAN STUURPOMP HYDRAULIEK ARM
ANDNOT 3380.11
LDNOT I_5WS15  ; WERKSCHAKELAAR AAN STUURPOMP HYDRAULIEK ARM
AND 3380.11
ORLD
ANDLD
TIM 0511 D20  ; `
AND T0511
SET H300.11

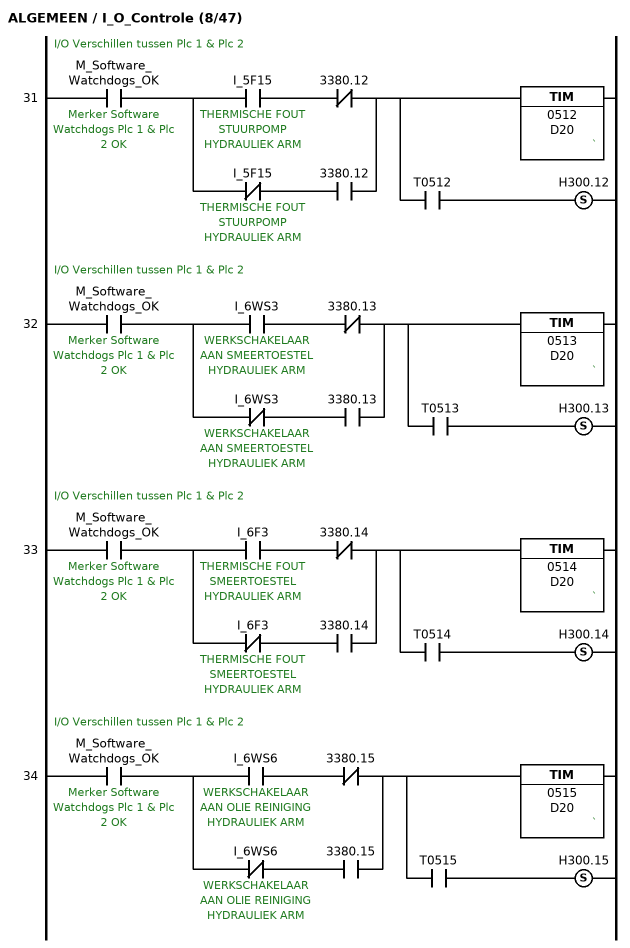
; rung 31: I/O Verschillen tussen Plc 1 & Plc 2
LD M_Software_Watchdogs_OK  ; Merker Software Watchdogs Plc 1 & Plc 2 OK
LD I_5F15  ; THERMISCHE FOUT STUURPOMP HYDRAULIEK ARM
ANDNOT 3380.12
LDNOT I_5F15  ; THERMISCHE FOUT STUURPOMP HYDRAULIEK ARM
AND 3380.12
ORLD
ANDLD
TIM 0512 D20  ; `
AND T0512
SET H300.12
; rung 32: I/O Verschillen tussen Plc 1 & Plc 2
LD M_Software_Watchdogs_OK  ; Merker Software Watchdogs Plc 1 & Plc 2 OK
LD I_6WS3  ; WERKSCHAKELAAR AAN SMEERTOESTEL HYDRAULIEK ARM
ANDNOT 3380.13
LDNOT I_6WS3  ; WERKSCHAKELAAR AAN SMEERTOESTEL HYDRAULIEK ARM
AND 3380.13
ORLD
ANDLD
TIM 0513 D20  ; `
AND T0513
SET H300.13
; rung 33: I/O Verschillen tussen Plc 1 & Plc 2
LD M_Software_Watchdogs_OK  ; Merker Software Watchdogs Plc 1 & Plc 2 OK
LD I_6F3  ; THERMISCHE FOUT SMEERTOESTEL HYDRAULIEK ARM
ANDNOT 3380.14
LDNOT I_6F3  ; THERMISCHE FOUT SMEERTOESTEL HYDRAULIEK ARM
AND 3380.14
ORLD
ANDLD
TIM 0514 D20  ; `
AND T0514
SET H300.14
; rung 34: I/O Verschillen tussen Plc 1 & Plc 2
LD M_Software_Watchdogs_OK  ; Merker Software Watchdogs Plc 1 & Plc 2 OK
LD I_6WS6  ; WERKSCHAKELAAR AAN OLIE REINIGING HYDRAULIEK ARM
ANDNOT 3380.15
LDNOT I_6WS6  ; WERKSCHAKELAAR AAN OLIE REINIGING HYDRAULIEK ARM
AND 3380.15
ORLD
ANDLD
TIM 0515 D20  ; `
AND T0515
SET H300.15

